PROGRAM MAIN_Motoransteuerung
VAR
	//Achsen Referenzen
	axis1: AXIS_REF;
	axis2: AXIS_REF;
	axis3: AXIS_REF;
	
	//Objekte um Achsen anzusteuern
	powerAxis1: MC_Power;
	driveAxis1: MC_MoveVelocity;
	driveAxis12: MC_MoveVelocity;
	resetAxis1: MC_Reset;
	
	powerAxis2: MC_Power;
	driveAxis2: MC_MoveVelocity;
	driveAxis22: MC_MoveVelocity;
	resetAxis2: MC_Reset;
	
	powerAxis3: MC_Power;
	driveAxis3: MC_MoveVelocity;
	driveAxis32: MC_MoveVelocity;
	resetAxis3: MC_Reset;
	
	//Achse Freischalten, Regler Freischalten
	enableControl: BOOL	:=0;
	enablePos: BOOL		:=0;
	enableNeg: BOOL		:=0;
	override:  LREAL	:=0;
	
	//Fahrbefehl Ausführen
	driveExecute: BOOL	:=0;
	
	//State Maschine
	nextState:EnumState	:=EnumState.init;
	state:EnumState		:=EnumState.init;
	switchDrive:INT		:=0;
	
	delay:TON;
	
	//Inputs
	velocityToMotors1 AT%I*: LREAL;
	velocityToMotors2 AT%I*: LREAL;
	velocityToMotors3 AT%I*: LREAL;
	directionToMotors1 AT%I*: INT;
	directionToMotors2 AT%I*: INT;
	directionToMotors3 AT%I*: INT;
	bumper	   AT%I*: BOOL;
END_VAR

axis1.ReadStatus();
axis2.ReadStatus();
axis3.ReadStatus();

//Zu Ersetzen mit SwitchCase
//powerAxis1(Axis:=axis1,Enable:=enableControl,Enable_Positive:=enablePos,Enable_Negative:=enableNeg,Override:=override);
//IF powerAxis1.Status THEN
//	moveAxis1(Axis:=axis1,Velocity:=250,Direction:=MC_Positive_Direction,Execute:=1,BufferMode:=MC_Buffered);
//END_IF
//Zu Ersetzen mit SwitchCase

CASE state OF
	EnumState.init:
		enableControl:=1;
		enablePos:=1;
		enableNeg:=1;
		override:=100;
		
		powerAxis1(Axis:=axis1,Enable:=enableControl,Enable_Positive:=enablePos,Enable_Negative:=enableNeg,Override:=override);
		powerAxis2(Axis:=axis2,Enable:=enableControl,Enable_Positive:=enablePos,Enable_Negative:=enableNeg,Override:=override);
		powerAxis3(Axis:=axis3,Enable:=enableControl,Enable_Positive:=enablePos,Enable_Negative:=enableNeg,Override:=override);
		IF (powerAxis1.Status AND powerAxis2.Status AND powerAxis3.Status) THEN	
			nextState:=EnumState.drive1; 
			driveExecute:=1;
		END_IF
		IF (powerAxis1.Error OR powerAxis2.Error OR powerAxis3.Error) THEN
			nextState:=EnumState.reset;
		END_IF
		
	EnumState.drive1:
	
		driveAxis1(Axis:=axis1,Velocity:=velocityToMotors1,Direction:=directionToMotors1,Execute:=driveExecute,BufferMode:=MC_Aborting);
		driveAxis2(Axis:=axis2,Velocity:=velocityToMotors2,Direction:=directionToMotors2,Execute:=driveExecute,BufferMode:=MC_Aborting);
		driveAxis3(Axis:=axis3,Velocity:=velocityToMotors3,Direction:=directionToMotors3,Execute:=driveExecute,BufferMode:=MC_Aborting);
		//delay(IN:=1,PT:=T#500MS);
		switchDrive:=switchDrive+1;
		
		IF (switchDrive=2) THEN
			switchDrive:=0;
			nextState:=EnumState.drive2;
			driveExecute:=0;
			driveAxis1(Axis:=axis1,Execute:=driveExecute);
			driveAxis2(Axis:=axis2,Execute:=driveExecute);
			driveAxis3(Axis:=axis3,Execute:=driveExecute);
			driveExecute:=1;
			delay(IN:=0);
		END_IF
		
		IF (powerAxis1.Error OR powerAxis2.Error OR powerAxis3.Error) THEN
			nextState:=EnumState.reset;
		END_IF
		
	EnumState.drive2:
	
		driveAxis1(Axis:=axis1,Velocity:=velocityToMotors1,Direction:=directionToMotors1,Execute:=driveExecute,BufferMode:=MC_Aborting);
		driveAxis2(Axis:=axis2,Velocity:=velocityToMotors2,Direction:=directionToMotors2,Execute:=driveExecute,BufferMode:=MC_Aborting);
		driveAxis3(Axis:=axis3,Velocity:=velocityToMotors3,Direction:=directionToMotors3,Execute:=driveExecute,BufferMode:=MC_Aborting);
		//delay(IN:=1,PT:=T#500MS);
		switchDrive:=switchDrive+1;
		
		IF (switchDrive=2) THEN
			switchDrive:=0;
			nextState:=EnumState.drive1;
			driveExecute:=0;
			driveAxis1(Axis:=axis1,Execute:=driveExecute);
			driveAxis2(Axis:=axis2,Execute:=driveExecute);
			driveAxis3(Axis:=axis3,Execute:=driveExecute);
			driveExecute:=1;
			//delay(IN:=0);
		END_IF
		IF (powerAxis1.Error OR powerAxis2.Error OR powerAxis3.Error OR bumper) THEN
			nextState:=EnumState.reset;
		END_IF	
	EnumState.reset:
	
		powerAxis1(Axis:=axis1,Enable:=0,Enable_Positive:=0,Enable_Negative:=0,Override:=0);
		powerAxis2(Axis:=axis1,Enable:=0,Enable_Positive:=0,Enable_Negative:=0,Override:=0);
		powerAxis3(Axis:=axis1,Enable:=0,Enable_Positive:=0,Enable_Negative:=0,Override:=0);
		driveAxis1(Axis:=axis1,Velocity:=0,Direction:=0,Execute:=0,BufferMode:=MC_Aborting);
		driveAxis2(Axis:=axis1,Velocity:=0,Direction:=0,Execute:=0,BufferMode:=MC_Aborting);
		driveAxis3(Axis:=axis1,Velocity:=0,Direction:=0,Execute:=0,BufferMode:=MC_Aborting);
	
		resetAxis1(Axis:=axis1,Execute:=1);
		resetAxis2(Axis:=axis2,Execute:=1);
		resetAxis3(Axis:=axis3,Execute:=1);
	
		IF (resetAxis1.Done AND resetAxis2.Done AND resetAxis3.Done) THEN
					;
				END_IF	
	ELSE
		nextState:=EnumState.reset;
END_CASE
state:=nextState;

END_PROGRAM

(* stored: Version 1.1.0.1, ProductVersion 3.1.4022.3
   POU MAIN_Motoransteuerung: Id {16a347dc-587d-4819-9a09-e734dabd6320}, SpecialFunc None *)
